{region '#Template'}
	{attribute 'Version' := '5.0.0.0'}
	{attribute 'Tags' := '"LCID": "1031", "Text": "Universal, Control, Monitoring"'}
	{attribute 'Tags' := '"LCID": "1033", "Text": "Universal, Control, Monitoring"'}
	{attribute 'Using' := '"Type": "Template", "URI": "EC_ID"'}
	{attribute 'Using' := '"Type": "Template", "URI": "BA2_Param"'}
	{attribute 'Description' := '"LCID": "1031", "Text": "Überwachung von Signalen"'}
	{attribute 'Description' := '"LCID": "1033", "Text": "Monitoring signals"'}
{endregion}
FUNCTION_BLOCK FB_BA_FdbAnalog EXTENDS FB_BA_View
VAR_INPUT
	bEn						: BOOL;	
	bCommand				: BOOL;	
	fIn							: REAL;	
END_VAR
VAR_OUTPUT
	bDst					: BOOL;
END_VAR
VAR_INPUT CONSTANT
	SwitchOnValue			: FB_BA_AV_Op;									 
	SwitchOffValue			: FB_BA_AV_Op;												  									
	DelayFeedback			: FB_BA_AV_Op;
	DelayInterruption		: FB_BA_AV_Op;						 									  	
	Dst						: FB_BA_BV;			
END_VAR	
VAR
	FixedLimit				: FB_BA_Swi2P;
	FdbCtrl					: FB_BA_FdbCtrlBinary;
END_VAR

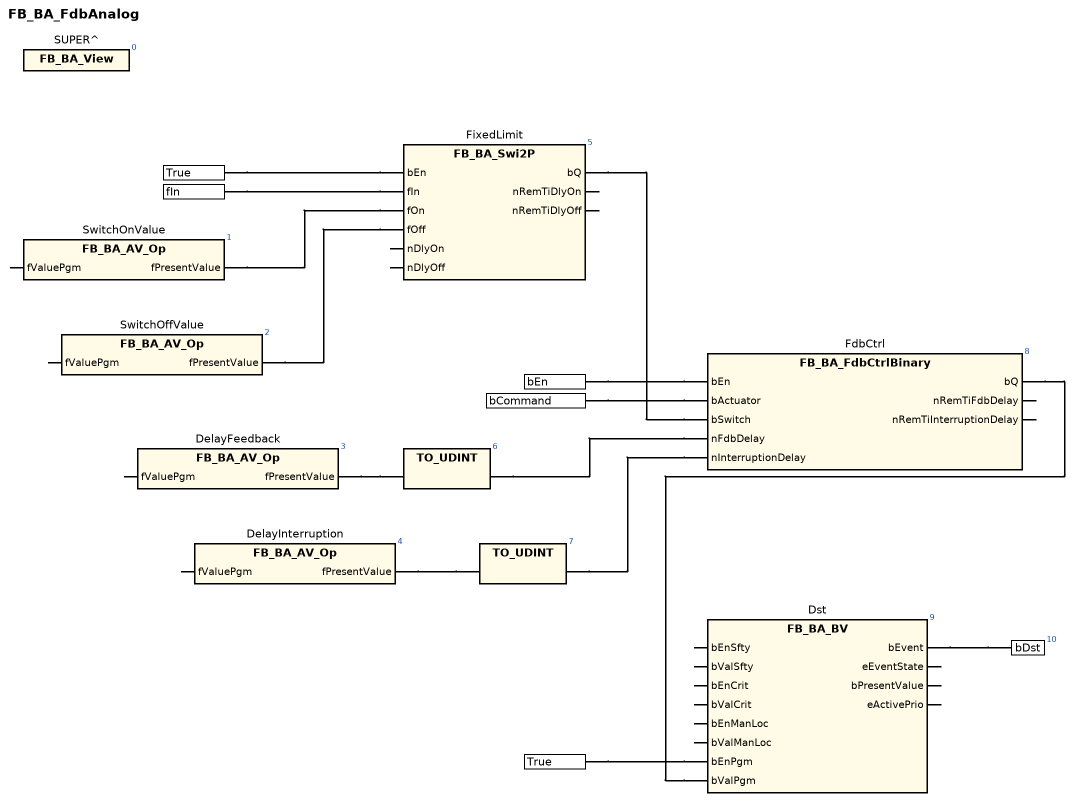
SUPER^(); // FB_BA_View
SwitchOnValue(); // FB_BA_AV_Op
SwitchOffValue(); // FB_BA_AV_Op
DelayFeedback(); // FB_BA_AV_Op
DelayInterruption(); // FB_BA_AV_Op
FixedLimit(bEn := True, fIn := fIn, fOn := SwitchOnValue.fPresentValue, fOff := SwitchOffValue.fPresentValue); // FB_BA_Swi2P
FdbCtrl(
    bEn := bEn,
    bActuator := bCommand,
    bSwitch := FixedLimit.bQ,
    nFdbDelay := TO_UDINT(DelayFeedback.fPresentValue),
    nInterruptionDelay := TO_UDINT(DelayInterruption.fPresentValue)); // FB_BA_FdbCtrlBinary
Dst(bEnPgm := True, bValPgm := FdbCtrl.bQ); // FB_BA_BV
bDst := Dst.bEvent;

METHOD FB_init : BOOL
VAR_INPUT
	bInitRetains : BOOL; // if TRUE, the retain variables are initialized (warm start / cold start)
	bInCopyCode : BOOL;  // if TRUE, the instance afterwards gets moved into the copy code (online change)
END_VAR
SwitchOnValue.iParent				:= THIS^;
SwitchOnValue.iLabel				:= LblFun_LimitMAX; 							 	 
SwitchOnValue.eUnit 				:= E_BA_Unit.ePressure_Pascals;								 
SwitchOnValue.fValueRm				:= 300;	
SwitchOnValue.fCOVIncrement			:= BA2_Param.fDefCOVIncrement;		
		
SwitchOffValue.iParent				:= THIS^;
SwitchOffValue.iLabel				:= LblFun_LimitMIN; 							 	 
SwitchOffValue.eUnit 				:= E_BA_Unit.ePressure_Pascals;								 
SwitchOffValue.fValueRm				:= 280;			
SwitchOffValue.fCOVIncrement		:= BA2_Param.fDefCOVIncrement;		

DelayFeedback.iParent				:= THIS^;
DelayFeedback.iLabel				:= LblFun_FeedbackDelay;							 	 
DelayFeedback.eUnit 				:= E_BA_Unit.eTime_Seconds;								 
DelayFeedback.fValueRm 				:= 120;
DelayFeedback.fCOVIncrement			:= BA2_Param.fDefCOVIncrement;		
							
DelayInterruption.iParent			:= THIS^;
DelayInterruption.iLabel			:= LblCtl_TimeDelayInterruptionFeedback;								 	 
DelayInterruption.eUnit 			:= E_BA_Unit.eTime_Seconds;								 
DelayInterruption.fValueRm 			:= 2;
DelayInterruption.fCOVIncrement		:= BA2_Param.fDefCOVIncrement;		
											 									  	
Dst.iParent							:= THIS^;
Dst.iLabel							:= LblFun_Fault; 
Dst.sActiveText 					:= txtEvent_Triggered;
Dst.sInactiveText 					:= txtEvent_Normal;
Dst.bEnManualRm						:= FALSE;	//	Priority  8	
Dst.bValManualRm					:= FALSE;	//	Priority  8
Dst.nEventClassID					:= EC_ID.NC30;
Dst.stTimeDelay.nToNormal			:= 0;
Dst.stTimeDelay.nToAbnormal			:= 0;
Dst.bAlarmValue						:= TRUE;
Dst.aEventTransitionText[1]			:= txtEvent_Triggered;
Dst.aEventTransitionText[2]			:= txtEvent_Error;
Dst.aEventTransitionText[3]			:= txtEvent_Normal;
Dst.bEventDetectionEnable			:= TRUE;
Dst.eEnPlantLock					:= E_BA_LockPriority.eNoLock;
END_METHOD

END_FUNCTION_BLOCK

(* stored: Version 1.1.0.1, ProductVersion 3.1.4024.12
   POU FB_BA_FdbAnalog: Id {1b70014a-31a0-491e-8162-8d5502a86e1a}, SpecialFunc None
   Method FB_init: Id {d1692fd2-ec24-4396-9cbc-e500bec0ff04} *)
